TYPE MaterialSlot :
STRUCT
	material : STRING;
	occupied AT %I* : BOOL;
END_STRUCT
END_TYPE

(* stored: Version 1.1.0.1, ProductVersion 3.1.4024.11
   DUT MaterialSlot: Id {346c1f05-ae71-4a21-928c-9d6ca77cc8a0} *)
